(* IEC 61131-3 sources: eCockpitGit/test_project/src/%F%00 Library/%F%Common Functions/%F%Math/%F%Rounding, 2 files *)

(* ---- %POU%FU_rCeiling.st ---- *)
//This function rounds the given value up to the nearest whole value
// |**Version**|**Author**| **Date** |**Changes**
// | 1         | NSN      | 18-05-22 | Creation
FUNCTION FU_rCeiling : REAL
VAR_INPUT
	rIn		:REAL;
END_VAR
(*%!%__DELIMITER__%!%*)
FU_rCeiling 	:=	TO_INT(rIn);
IF FU_rCeiling < rIn THEN
	FU_rCeiling := FU_rCeiling + 1;
END_IF;

(* ---- %POU%FU_rRound.st ---- *)
//This function rounds the input down to the amount of decimals inputted on iN
// |**Version**|**Author**| **Date** |**Changes**
// | 1         | NSN      | 11-03-19 | Creation
FUNCTION FU_rRound : REAL
VAR_INPUT
	X		:REAL;	//Value to be rounded
	N		:BYTE;	//Amount of decimals
END_VAR
(*%!%__DELIMITER__%!%*)
FU_bMinMaxValue(Variable:= N, MinVal:= 0, MaxVal:= 8);
FU_rRound := DINT_TO_REAL(REAL_TO_DINT(X * GConstants.exponents[N])) / GConstants.exponents[N];
